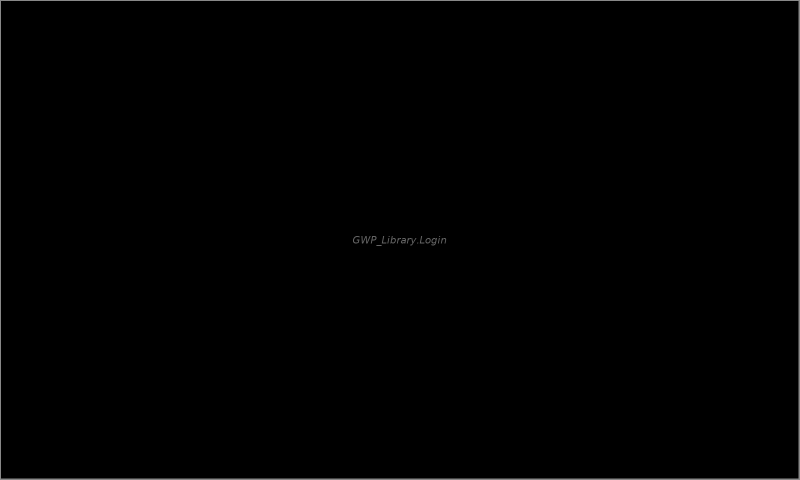
VISUALIZATION Login  // 800x480
    Frame (0,0 800x480)
        shows GWP_Library.Login(FB_Init_1 := Main.Init_0)
END_VISUALIZATION

(* stored: Version 1.1.0.1, ProductVersion 3.1.4022.6
   Visu Login: Id {fb49d956-77f2-414e-84df-6d301a67978d} *)
